FUNCTION TryConvert_INT_TO_BOOL : BOOL
VAR_INPUT
	in : INT;
	out : REFERENCE TO BOOL;
END_VAR

out := INT_TO_BOOL(in);
TryConvert_INT_TO_BOOL := TRUE;

END_FUNCTION

(* stored: Version 1.1.0.1, ProductVersion 3.1.4024.12
   POU TryConvert_INT_TO_BOOL: Id {d914834d-c802-4b5b-ac4c-38ad19b2b0a2}, SpecialFunc None *)
